# EPICS autosave request: GALIL/iocBoot/iocGALIL-IOC-01/IMATStagesMenu.req
file configMenu.req P=$(CMP),CONFIG=$(CONFIG)
file $(IOCNAME)_settings.req P=$(P),CCP=$(MTRCTRL)
